PROGRAM PiezoSerial
VAR
	//PI Serial
	fbE621SerialDriver_M1L0 : FB_PI_E621_SerialDriver;
	rtInitParams_M1L0	:	R_TRIG;
	tonTimeoutRst_M1L0	: TON := (PT:=T#2S); //For timeout reset
	
	fbE621SerialDriver_M2L0 : FB_PI_E621_SerialDriver;
	rtInitParams_M2L0	:	R_TRIG;
	tonTimeoutRst_M2L0	: TON := (PT:=T#2S); //For timeout reset
END_VAR

//Piezo E-621
///////////////////////
fbE621SerialDriver_M1L0.i_xExecute := TRUE;
fbE621SerialDriver_M1L0.i_xExecute R= fbE621SerialDriver_M1L0.q_xDone;
fbE621SerialDriver_M1L0(iq_stPiezoAxis:= GVL_M1L0.M1L0_Pitch.Piezo,
		                iq_stSerialRXBuffer:= Serial_RXBuffer_M1L0,
		                iq_stSerialTXBuffer:= Serial_TXBuffer_M1L0);

fbE621SerialDriver_M2L0.i_xExecute := TRUE;
fbE621SerialDriver_M2L0.i_xExecute R= fbE621SerialDriver_M2L0.q_xDone;
fbE621SerialDriver_M2L0(iq_stPiezoAxis:= M2L0_Pitch.Piezo,
		                iq_stSerialRXBuffer:= Serial_RXBuffer_M2L0,
		                iq_stSerialTXBuffer:= Serial_TXBuffer_M2L0);

END_PROGRAM

(* stored: Version 1.1.0.1, ProductVersion 3.1.4022.18
   POU PiezoSerial: Id {04ed9258-9624-4f29-9f34-d3e5ff9995d6}, SpecialFunc None *)
